PROGRAM PLC_PRG
VAR
	//Visualization buttons
	mxButtonStart: BOOL;	
	mxButtonReset: BOOL;
	
	//Intarnal use
	mxComBusy: BOOL;
	mxDone: BOOL;
	mxStart: BOOL;
	ComData: CommunicationData;	

	//Motion function blocks
	fbCommunicator: Communicator;
	fbABBGoToHome_1: ABBGoToHome;

	fbABBGoToStorage_1: ABBGoToStorage;
	fbABBPickLeaveStorage_1: ABBPickLeaveStorage;
END_VAR

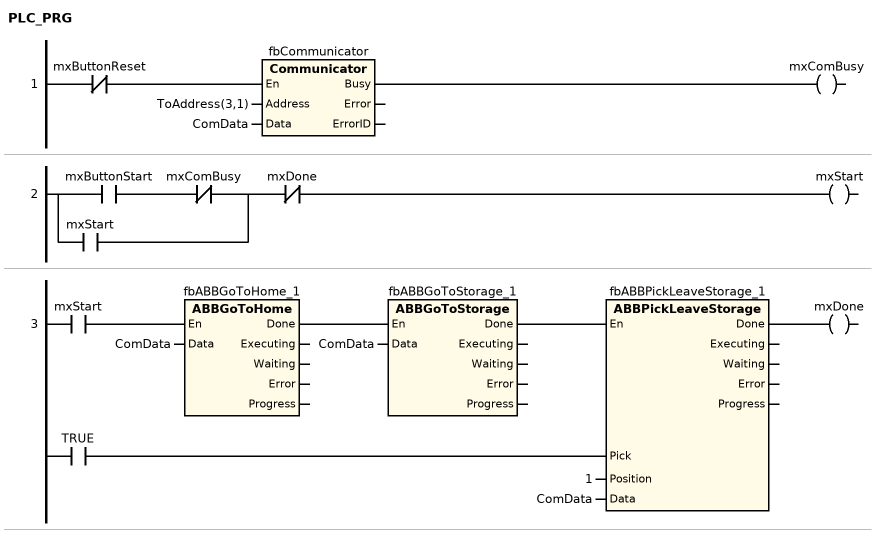
// NETWORK 1
fbCommunicator(En := NOT mxButtonReset, Address := ToAddress(3,1), Data := ComData); // Communicator
mxComBusy := fbCommunicator.Busy;

// NETWORK 2
mxStart := (mxButtonStart AND NOT mxComBusy OR mxStart) AND NOT mxDone;

// NETWORK 3
fbABBGoToHome_1(En := mxStart, Data := ComData); // ABBGoToHome
fbABBGoToStorage_1(En := fbABBGoToHome_1.Done, Data := ComData); // ABBGoToStorage
fbABBPickLeaveStorage_1(En := fbABBGoToStorage_1.Done, Pick := TRUE, Position := 1, Data := ComData); // ABBPickLeaveStorage
mxDone := fbABBPickLeaveStorage_1.Done;

END_PROGRAM

(* stored: Version 1.1.0.1, ProductVersion 3.1.4022.12
   POU PLC_PRG: Id {ac26337c-3067-480e-ac28-5dd5bee58459}, SpecialFunc None *)
